Universal Robots PolyScope program: point.urp

Program point (installation=uwaur5 directory=/programs createdIn=3.10.1.76190 lastSavedIn=3.10.1.76190 robotSerialNumber=2017356443)
Calibrated DH parameters: a=[0.000092, -0.116521, -0.182101, -0.000106, 0.000044, 0]; d=[0.089391, 255.189113, -82.629387, -172.449369, 0.094782, 0.082637]; alpha=[1.569598, 0.001603, 0.002015, 1.570234, -1.570307, 0]; deltaTheta=[-0.000017, 1.293309, -0.204843, -1.088417, 0.000036, -0.000078]
Robot Program (runOnlyOnce=false)
  Set NoAction
  MoveJ speed 60 deg/s, acceleration 80 deg/s^2 (useActiveTCP=true)
    Waypoint Waypoint_1: TCP in base x=600.728 y=-63.396 z=284.57 mm, rx=-2.1697 ry=2.1838 rz=0.0067 rad; joints [4.227, -107.333, -92.422, -67.694, 92.623, 4.501] deg
  Set NoAction
  MoveJ speed 60 deg/s, acceleration 80 deg/s^2 (useActiveTCP=true)
    Waypoint Waypoint_2: TCP in base x=292.177 y=-85.857 z=690.733 mm, rx=-1.9926 ry=1.9904 rz=-0.2922 rad; joints [4.205, -70.611, -71.124, -107.139, 92.678, 4.498] deg
      Until NONE (allowActions=false)
    URCap Gripper (Robotiq_2-Finger_Adaptive_Gripper, Robotiq Inc.)
    URCap Cam Locate (Robotiq_Wrist_Camera, Robotiq Inc.)
      Placeholder
